Xinje XCPPro project, PLC1: XC3-24 (software 3.3q)

PROGRAM Ladder

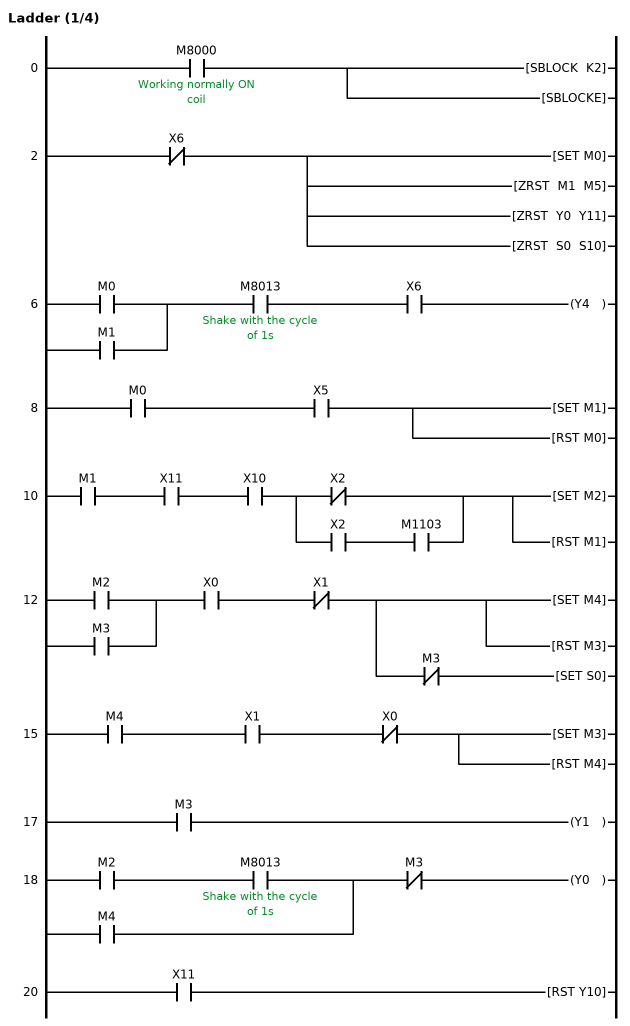
LD     M8000	; Working normally ON coil
SBLOCK K2
SBLOCKE
LDI    X6
SET    M0
ZRST   M1 M5
ZRST   Y0 Y11
ZRST   S0 S10
LD     M0
OR     M1
AND    M8013	; Shake with the cycle of 1s
AND    X6
OUT    Y4
LD     M0
AND    X5
SET    M1
RST    M0
LD     M1
AND    X11
AND    X10
LDI    X2
LD     X2
AND    M1103
ORB
ANB
SET    M2
RST    M1
LD     M2
OR     M3
AND    X0
ANI    X1
SET    M4
RST    M3
ANI    M3
SET    S0
LD     M4
AND    X1
ANI    X0
SET    M3
RST    M4
LD     M3
OUT    Y1
LD     M2
AND    M8013	; Shake with the cycle of 1s
OR     M4
ANI    M3
OUT    Y0
LD     X11
RST    Y10

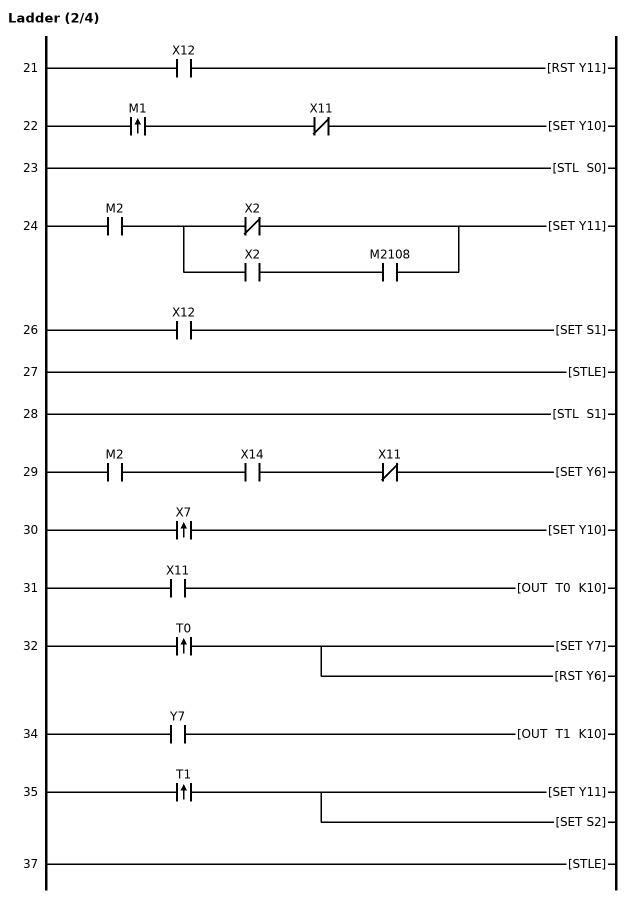
LD     X12
RST    Y11
LDP    M1
ANI    X11
SET    Y10
STL    S0
LD     M2
LDI    X2
LD     X2
AND    M2108
ORB
ANB
SET    Y11
LD     X12
SET    S1
STLE
STL    S1
LD     M2
AND    X14
ANI    X11
SET    Y6
LDP    X7
SET    Y10
LD     X11
OUT    T0 K10
LDP    T0
SET    Y7
RST    Y6
LD     Y7
OUT    T1 K10
LDP    T1
SET    Y11
SET    S2
STLE

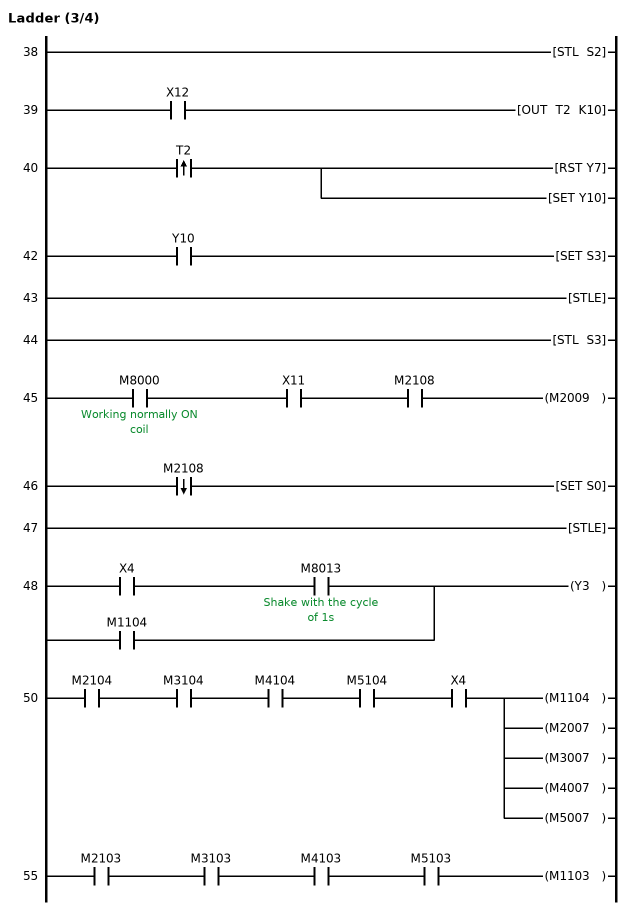
STL    S2
LD     X12
OUT    T2 K10
LDP    T2
RST    Y7
SET    Y10
LD     Y10
SET    S3
STLE
STL    S3
LD     M8000	; Working normally ON coil
AND    X11
AND    M2108
OUT    M2009
LDF    M2108
SET    S0
STLE
LD     X4
AND    M8013	; Shake with the cycle of 1s
OR     M1104
OUT    Y3
LD     M2104
AND    M3104
AND    M4104
AND    M5104
AND    X4
OUT    M1104
OUT    M2007
OUT    M3007
OUT    M4007
OUT    M5007
LD     M2103
AND    M3103
AND    M4103
AND    M5103
OUT    M1103

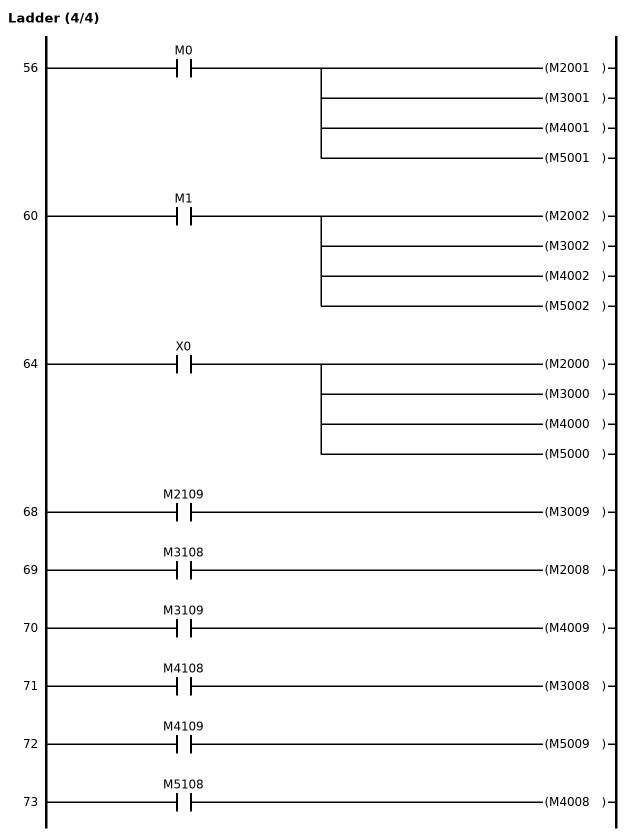
LD     M0
OUT    M2001
OUT    M3001
OUT    M4001
OUT    M5001
LD     M1
OUT    M2002
OUT    M3002
OUT    M4002
OUT    M5002
LD     X0
OUT    M2000
OUT    M3000
OUT    M4000
OUT    M5000
LD     M2109
OUT    M3009
LD     M3108
OUT    M2008
LD     M3109
OUT    M4009
LD     M4108
OUT    M3008
LD     M4109
OUT    M5009
LD     M5108
OUT    M4008